FUNCTION_BLOCK E_RESTART
  (* Version 1.0, 2005-04-08, Goran Cengic, Chalmers *)
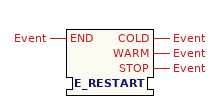
  EVENT_INPUT
    END;
  END_EVENT
  EVENT_OUTPUT
    COLD;
    WARM;
    STOP;
  END_EVENT
END_FUNCTION_BLOCK
